(* PLC project po, TNI-Software ControlBuild 4.00 *)
(* stored: creationDateTime 2018-09-17T17:25:09-01:00 *)

PROGRAM tapis_conv.po
  VAR_INPUT  (* CB.group=Commande_PO CB.kind=inputVars *)
    Marche : BOOL := false;
  END_VAR
  VAR_INPUT  (* CB.group=Retour_Utilisateur CB.kind=inputVars *)
    Chargement : BOOL := false;
    Dechargement : BOOL := false;
  END_VAR
  VAR_OUTPUT  (* CB.group=Retour_PO CB.kind=outputVars *)
    Fin_Convoyage : BOOL := false;
  END_VAR

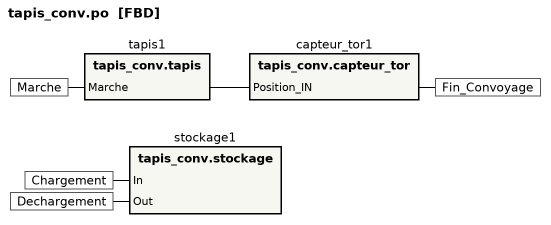
(* FBD diagram, written out as Structured Text *)
tapis1(Marche := Marche);
capteur_tor1(Position_IN := tapis1.Deplacement);
Fin_Convoyage := capteur_tor1.Etat;
stockage1(In := Chargement, Out := Dechargement);
END_PROGRAM
